{attribute 'qualified_only'}
VAR_GLOBAL CONSTANT
	MAX_LICZBA_PODZESPOLOW					: int := 10;
END_VAR

(* stored: Version 1.1.0.1, ProductVersion 3.1.4024.11
   GVL GVL_StanMaszyny_STALE: Id {155edd62-d26a-4311-86c8-ceedafb0660a} *)
